// Mitsubishi GX Works2 project: 0709   PLC: Q02/Q02H

PROGRAM MAIN
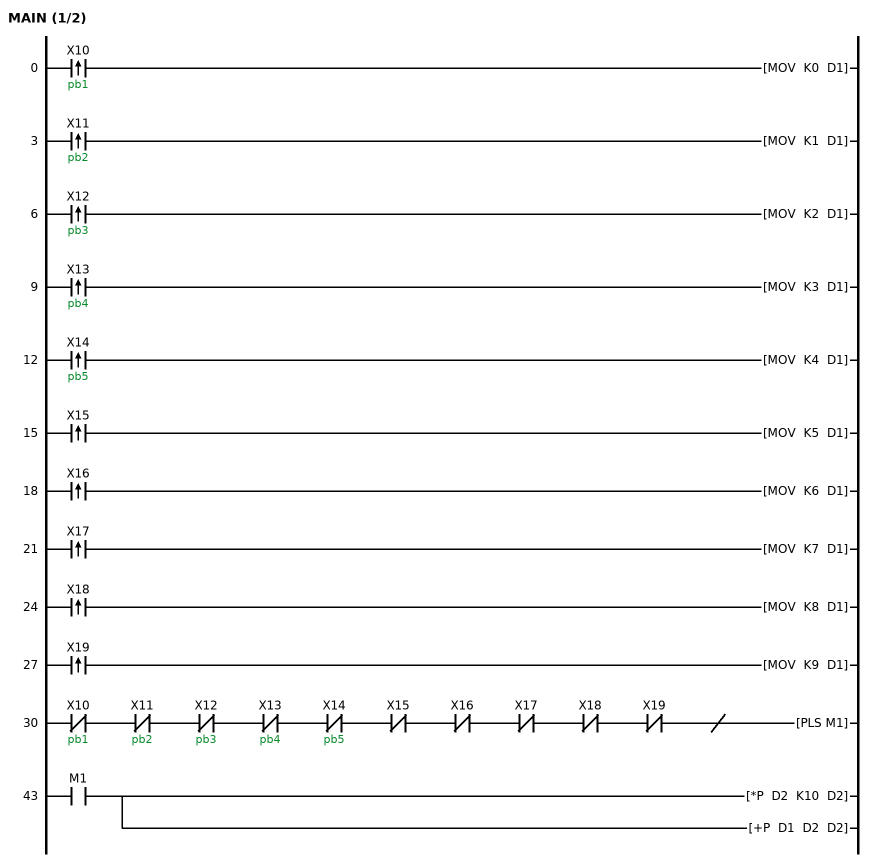
0     LDP     X10  ; pb1
      MOV     K0 D1
3     LDP     X11  ; pb2
      MOV     K1 D1
6     LDP     X12  ; pb3
      MOV     K2 D1
9     LDP     X13  ; pb4
      MOV     K3 D1
12    LDP     X14  ; pb5
      MOV     K4 D1
15    LDP     X15
      MOV     K5 D1
18    LDP     X16
      MOV     K6 D1
21    LDP     X17
      MOV     K7 D1
24    LDP     X18
      MOV     K8 D1
27    LDP     X19
      MOV     K9 D1
30    LDI     X10  ; pb1
      ANI     X11  ; pb2
      ANI     X12  ; pb3
      ANI     X13  ; pb4
      ANI     X14  ; pb5
      ANI     X15
      ANI     X16
      ANI     X17
      ANI     X18
      ANI     X19
      INV
      PLS     M1
43    LD      M1
      *P      D2 K10 D2
      +P      D1 D2 D2
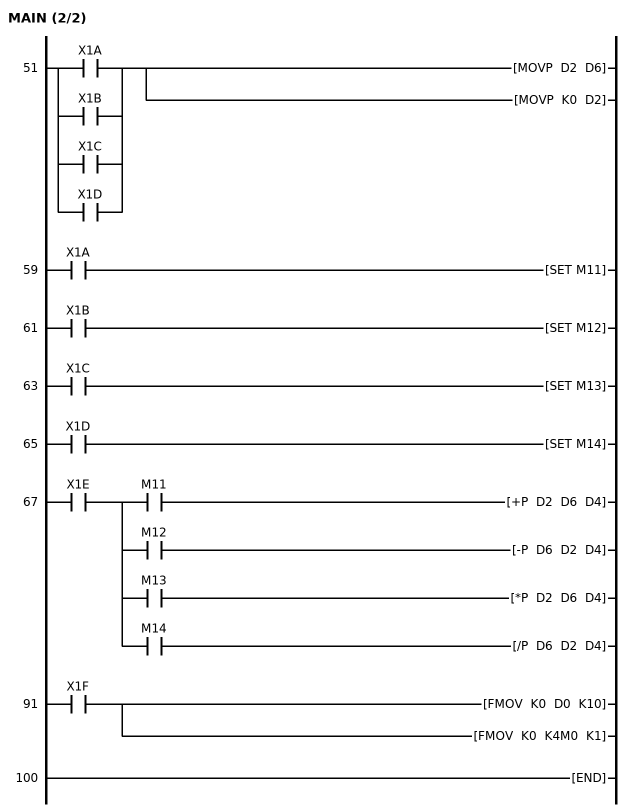
51    LD      X1A
      OR      X1B
      OR      X1C
      OR      X1D
      MOVP    D2 D6
      MOVP    K0 D2
59    LD      X1A
      SET     M11
61    LD      X1B
      SET     M12
63    LD      X1C
      SET     M13
65    LD      X1D
      SET     M14
67    LD      X1E
      MPS
      AND     M11
      +P      D2 D6 D4
      MRD
      AND     M12
      -P      D6 D2 D4
      MRD
      AND     M13
      *P      D2 D6 D4
      MPP
      AND     M14
      /P      D6 D2 D4
91    LD      X1F
      FMOV    K0 D0 K10
      FMOV    K0 K4M0 K1
100   END
END_PROGRAM

PROGRAM sub1
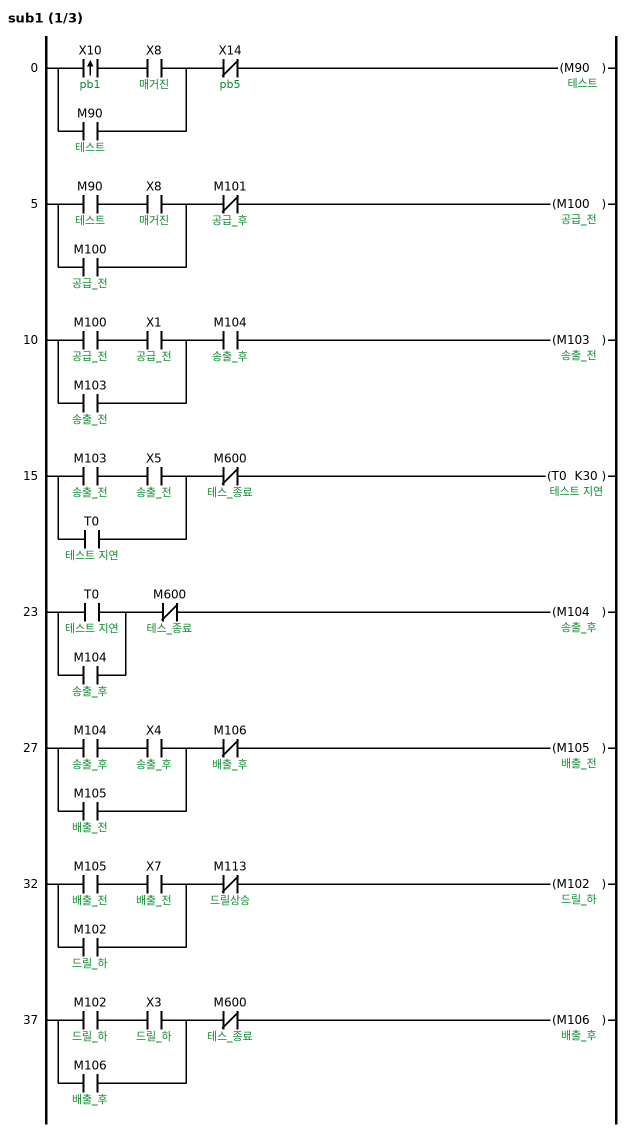
0     LDP     X10  ; pb1
      AND     X8  ; 매거진
      OR      M90  ; 테스트
      ANI     X14  ; pb5
      OUT     M90  ; 테스트
5     LD      M90  ; 테스트
      AND     X8  ; 매거진
      OR      M100  ; 공급_전
      ANI     M101  ; 공급_후
      OUT     M100  ; 공급_전
10    LD      M100  ; 공급_전
      AND     X1  ; 공급_전
      OR      M103  ; 송출_전
      AND     M104  ; 송출_후
      OUT     M103  ; 송출_전
15    LD      M103  ; 송출_전
      AND     X5  ; 송출_전
      OR      T0  ; 테스트 지연
      ANI     M600  ; 테스_종료
      OUT     T0 K30  ; 테스트 지연
23    LD      T0  ; 테스트 지연
      OR      M104  ; 송출_후
      ANI     M600  ; 테스_종료
      OUT     M104  ; 송출_후
27    LD      M104  ; 송출_후
      AND     X4  ; 송출_후
      OR      M105  ; 배출_전
      ANI     M106  ; 배출_후
      OUT     M105  ; 배출_전
32    LD      M105  ; 배출_전
      AND     X7  ; 배출_전
      OR      M102  ; 드릴_하
      ANI     M113  ; 드릴상승
      OUT     M102  ; 드릴_하
37    LD      M102  ; 드릴_하
      AND     X3  ; 드릴_하
      OR      M106  ; 배출_후
      ANI     M600  ; 테스_종료
      OUT     M106  ; 배출_후
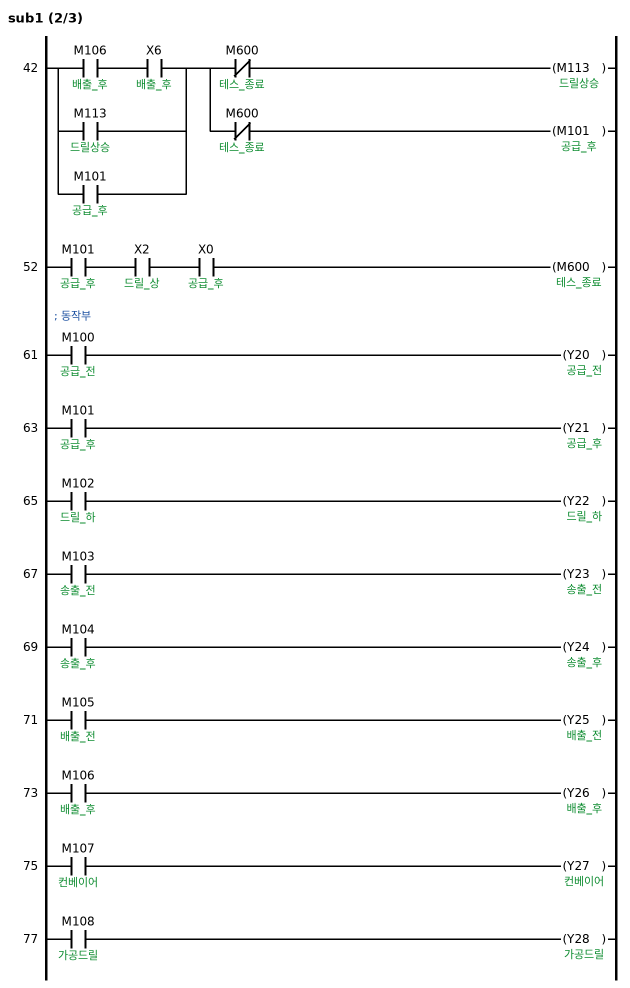
42    LD      M106  ; 배출_후
      AND     X6  ; 배출_후
      OR      M113  ; 드릴상승
      OR      M101  ; 공급_후
      MPS
      ANI     M600  ; 테스_종료
      OUT     M113  ; 드릴상승
      MPP
      ANI     M600  ; 테스_종료
      OUT     M101  ; 공급_후
52    LD      M101  ; 공급_후
      AND     X2  ; 드릴_상
      AND     X0  ; 공급_후
      OUT     M600  ; 테스_종료
; 동작부
61    LD      M100  ; 공급_전
      OUT     Y20  ; 공급_전
63    LD      M101  ; 공급_후
      OUT     Y21  ; 공급_후
65    LD      M102  ; 드릴_하
      OUT     Y22  ; 드릴_하
67    LD      M103  ; 송출_전
      OUT     Y23  ; 송출_전
69    LD      M104  ; 송출_후
      OUT     Y24  ; 송출_후
71    LD      M105  ; 배출_전
      OUT     Y25  ; 배출_전
73    LD      M106  ; 배출_후
      OUT     Y26  ; 배출_후
75    LD      M107  ; 컨베이어
      OUT     Y27  ; 컨베이어
77    LD      M108  ; 가공드릴
      OUT     Y28  ; 가공드릴
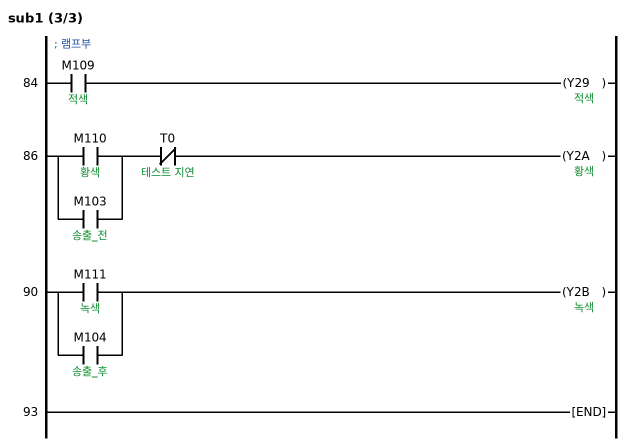
; 램프부
84    LD      M109  ; 적색
      OUT     Y29  ; 적색
86    LD      M110  ; 황색
      OR      M103  ; 송출_전
      ANI     T0  ; 테스트 지연
      OUT     Y2A  ; 황색
90    LD      M111  ; 녹색
      OR      M104  ; 송출_후
      OUT     Y2B  ; 녹색
93    END
END_PROGRAM

// device comments not shown above
X9  ; 비금속
X0A  ; 금속
M91  ; 단속
M92  ; 연속
M93  ; 초기화
M94  ; 종료1
M95  ; 종료2
M112  ; 드릴정지
M114  ; 금속탐지
M115  ; 비금속탐지
M200  ; 공급_전2
M201  ; 공급_후2
M202  ; 드릴_하2
M203  ; 송출_전2
M204  ; 송출_후2
M205  ; 배출_전2
M206  ; 배출_후2
M207  ; 컨베이어
M208  ; 가공드릴2
M209  ; 적색2
M210  ; 황색2
M211  ; 녹색2
M212  ; 드릴정지2
M213  ; 드릴상승2
M214  ; 금속탐지2
M215  ; 비금속탐지2
M300  ; 공급_전3
M301  ; 공급_후3
M302  ; 드릴_하3
M303  ; 송출_전3
M304  ; 송출_후3
M305  ; 배출_전3
M306  ; 배출_후3
M307  ; 컨베이어3
M308  ; 가공드릴3
M309  ; 적색3
M310  ; 황색3
M311  ; 녹색3
M312  ; 드릴정지3
M313  ; 드릴상승3
M314  ; 금속탐지3
M315  ; 비금속탐지3
M400  ; 공급_전4
M401  ; 공급_후4
M402  ; 드릴_하4
M403  ; 송출_전4
M404  ; 송출_후4
M405  ; 배출_전4
M406  ; 배출_후4
M407  ; 컨베이어4
M408  ; 가공드릴4
M409  ; 적색4
M410  ; 황색4
M411  ; 녹색4
M412  ; 드릴정지4
M413  ; 드릴상승4
M414  ; 금속탐지4
M415  ; 비금속탐지4
M500  ; 금속1
M501  ; 금속2
M601  ; 종료1
M602  ; 종료2
M603  ; 종료3
M604  ; 종료4
T10  ; 금속지연
T11  ; 비금속지연
T20  ; 금속지연
T21  ; 비금속지연
T30  ; 비상 지연
